FUNCTION_BLOCK VisionCmdProcessor EXTENDS Module
VAR_INPUT
	Command: STRING(GVL.COMMAND_LEN) := '';
	LogicCmdIO: REFERENCE TO ST_LogicCmdIO;
	VisionSystemIpAddress: STRING(19) := '127.0.0.1';
	VisionSystemPort: UINT := 50011;
END_VAR
VAR_OUTPUT
	VisionStateText: STRING := 'READY';
END_VAR
VAR
	_CaptureImage_Output: STRING(255);
	_CaptureImage_WorkerUid: STRING;
	_LocatePart_Output: STRING(255);
	_LocatePart_WorkerUid: STRING;
	_RunCalibration_Output: STRING(255);
	_RunCalibration_WorkerUid: STRING;
	_Vision: OpenCV;
	_VisionCommandParser: ParseVisionCmd;
	_VisionDoneRtrig: R_TRIG;
	_VisionBusyRtrig: R_TRIG;
	_VisionResult: STRING(255);
	_ResultPosition: INT;
	_ResultPosition_CAL: INT;
	_ResultPosition_LOC: INT;
	_ResultPosition_CAP: INT;
	_SpacePosition: INT;
	_VisionObjectIndex: UINT;
	_VisionRatio: REAL;
	_VisionRotation: REAL;
	_VisionError: REAL;
	_PartsCount: UDINT;
	_UnitModeCurrentState: PACK_ML.State;
END_VAR
VAR CONSTANT
	_RESPONSE_CAL: STRING := 'res: CAL ';
	_RESPONSE_LOC: STRING := 'res: LOC ';
	_RESPONSE_CAP: STRING := 'res: CAP ';
	_STEP_DONE: INT := 1000;
	_STEP_IDLE: INT := 0;
	_STEP_COMMAND: INT := 20;
	_STEP_TRIGGER: INT := 30;
	_STEP_WAIT: INT := 40;
	_STEP_ERR: INT := 50;
END_VAR

SUPER^();

// PackML state machine implementation
_UnitModeCurrentState := SUPER^._UnitMode.CurrentState;

//
CASE SUPER^._SeqMain OF
	
    _STEP_DONE:
		SUPER^._SeqMain := _STEP_IDLE;
        
    _STEP_IDLE:
		// hang out here until called to run
        
    _STEP_COMMAND: // parse vision command
        _VisionCommandParser(Command:=Command);
		IF _VisionCommandParser.Error THEN
			SUPER^.M_Error(Description:=_VisionCommandParser.ErrorDescription);
			//
			SUPER^._SeqMain := _STEP_ERR;
		ELSE
			IF _VisionCommandParser.stCommand.Timeout > 0 THEN
				SUPER^._TimeoutTimer.PT := UDINT_TO_TIME(_VisionCommandParser.stCommand.Timeout * 1000);
			END_IF
			//
			SUPER^._SeqMain := _STEP_TRIGGER;
		END_IF
		
	_STEP_TRIGGER: //
		CASE _VisionCommandParser.stCommand.CommandType OF
			DUT_Command_VisionType.Calibrate: //
				_Vision.M_CalibrateCamera(	iImageWidth:= _VisionCommandParser.stCommand.ImageWidth, 
											iImageHeight:= _VisionCommandParser.stCommand.ImageHeight, 
											fCalCheckerSize:= _VisionCommandParser.stCommand.Calibrate.CheckerSize, 
											iCalCheckerX:= _VisionCommandParser.stCommand.Calibrate.CheckerXCount, 
											iCalCheckerY:= _VisionCommandParser.stCommand.Calibrate.CheckerYCount,
                                            uTimeout:=_VisionCommandParser.stCommand.Timeout);
			
			DUT_Command_VisionType.Acquire: //
				_Vision.M_CaptureImage(	iImageWidth:= _VisionCommandParser.stCommand.ImageWidth, 
										iImageHeight:= _VisionCommandParser.stCommand.ImageHeight,
                                        uTimeout:=_VisionCommandParser.stCommand.Timeout);
			
			DUT_Command_VisionType.LocatePart: //
				_PartsCount := 0;
				LogicCmdIO.Register[_VisionCommandParser.stCommand.Locate.ResultPosition] := 0;
				_Vision.M_LocatePart( 	iImageWidth:= _VisionCommandParser.stCommand.ImageWidth, 
										iImageHeight:= _VisionCommandParser.stCommand.ImageHeight, 
										iMaxPos:= _VisionCommandParser.stCommand.Locate.MaxParts, 
										dMaxOverlap:= _VisionCommandParser.stCommand.Locate.MaxOverlap, 
										dScore:= _VisionCommandParser.stCommand.Locate.Score, 
										dToleranceAngle:= _VisionCommandParser.stCommand.Locate.ToleranceAngle,
                                        uTimeout:=_VisionCommandParser.stCommand.Timeout,
										sTemplateName:=_VisionCommandParser.stCommand.Locate.TemplateName,
										sScriptFilename:=_VisionCommandParser.stCommand.Locate.ScriptFilename);
			
		END_CASE;
		
		//
		SUPER^._SeqMain := _STEP_WAIT;
		
	_STEP_WAIT: //
		IF _VisionDoneRtrig.Q THEN
			
			//
			_VisionResult := _Vision.P_Response;
			
			//
			_ResultPosition_CAL := FIND(STR1:=_VisionResult,STR2:=_RESPONSE_CAL);
			_ResultPosition_LOC := FIND(STR1:=_VisionResult,STR2:=_RESPONSE_LOC);
			_ResultPosition_CAP := FIND(STR1:=_VisionResult,STR2:=_RESPONSE_CAP);
			
			//
			IF _ResultPosition_CAL > 0 THEN 
				// calibration was completed
				// res: CAL rat:23.23 rot:23.23 err:23.23
				_VisionResult := MID(STR:=_VisionResult,LEN:=LEN(_VisionResult)-LEN(_RESPONSE_CAL),POS:=LEN(_RESPONSE_CAL)+1);
				//VisionStateText := CONCAT(VisionStateText, '\n');
				//VisionStateText := CONCAT(VisionStateText, _VisionResult);
				// rat:23.23 rot:23.23 err:23.23
				_ResultPosition := FIND(STR1:=_VisionResult,STR2:='rat:');
				IF _ResultPosition > 0 THEN
					_VisionResult := MID(STR:=_VisionResult,LEN:=LEN(_VisionResult)-LEN('rat:'),POS:=LEN('rat:')+1);
					_SpacePosition := FIND(STR1:=_VisionResult,STR2:=' ');
					_VisionRatio := STRING_TO_REAL(MID(STR:=_VisionResult,LEN:=_SpacePosition-1,POS:=1));
					_VisionResult := MID(STR:=_VisionResult,LEN:=LEN(_VisionResult)-_SpacePosition,POS:=_SpacePosition+1);
				END_IF
				// rot:23.23 err:23.23
				_ResultPosition := FIND(STR1:=_VisionResult,STR2:='rot:');
				IF _ResultPosition > 0 THEN
					_VisionResult := MID(STR:=_VisionResult,LEN:=LEN(_VisionResult)-LEN('rot:'),POS:=LEN('rot:')+1);
					_SpacePosition := FIND(STR1:=_VisionResult,STR2:=' ');
					_VisionRotation := STRING_TO_REAL(MID(STR:=_VisionResult,LEN:=_SpacePosition-1,POS:=1));
					_VisionResult := MID(STR:=_VisionResult,LEN:=LEN(_VisionResult)-_SpacePosition,POS:=_SpacePosition+1);
				END_IF
				// err:23.23
				_ResultPosition := FIND(STR1:=_VisionResult,STR2:='err:');
				IF _ResultPosition > 0 THEN
					_VisionResult := MID(STR:=_VisionResult,LEN:=LEN(_VisionResult)-LEN('err:'),POS:=LEN('err:')+1);
					_SpacePosition := FIND(STR1:=_VisionResult,STR2:=' ');
					_VisionError := STRING_TO_REAL(MID(STR:=_VisionResult,LEN:=_SpacePosition-1,POS:=1));
					_VisionResult := MID(STR:=_VisionResult,LEN:=LEN(_VisionResult)-_SpacePosition,POS:=_SpacePosition+1);
				END_IF
				
			ELSIF _ResultPosition_LOC > 0 THEN 
				// part was located
				// 'res: LOC obj:0 cx:54.66 cy:119.45 a:-12.87 s:0.84 $NLOC obj:1 cx:71.49 cy:100.06 a:10.13 s:0.83 $N'
				_VisionResult := MID(STR:=_VisionResult,LEN:=LEN(_VisionResult)-LEN(_RESPONSE_LOC),POS:=LEN(_RESPONSE_LOC)+1);
				//VisionStateText := CONCAT(VisionStateText, '\n');
				//VisionStateText := CONCAT(VisionStateText, _VisionResult);
				_VisionObjectIndex := 0;
				WHILE FIND(STR1:=_VisionResult,STR2:='obj:') > 0 
					AND _VisionObjectIndex <= _VisionCommandParser.stCommand.Locate.MaxParts 
					AND _VisionObjectIndex + _VisionCommandParser.stCommand.Locate.ResultPosition < GVL.VIS_ARR_END DO
					// 'obj:0 cx:54.66 cy:119.45 a:-12.87 s:0.84 $NLOC obj:1 cx:71.49 cy:100.06 a:10.13 s:0.83 $N'
					// $NLOC obj:1 cx:71.49 cy:100.06 a:10.13 s:0.83 $N'
					_ResultPosition := FIND(STR1:=_VisionResult,STR2:='obj:');
					IF _ResultPosition > 0 THEN
						_PartsCount := _PartsCount + 1;
						_VisionResult := MID(STR:=_VisionResult,LEN:=LEN(_VisionResult)-_ResultPosition-LEN('obj:')+1,POS:=_ResultPosition+LEN('obj:'));
						_SpacePosition := FIND(STR1:=_VisionResult,STR2:=' ');
						_VisionObjectIndex := STRING_TO_UINT(MID(STR:=_VisionResult,LEN:=_SpacePosition-1,POS:=1));
						SUPER^.VisionRegisters[_VisionCommandParser.stCommand.Locate.ResultPosition + _VisionObjectIndex].Comment := CONCAT('obj:', UDINT_TO_STRING(_VisionObjectIndex));
						_VisionResult := MID(STR:=_VisionResult,LEN:=LEN(_VisionResult)-_SpacePosition,POS:=_SpacePosition+1);
					END_IF
					// cx:54.66 cy:119.45 a:-12.87 s:0.84 $NLOC obj:1 cx:71.49 cy:100.06 a:10.13 s:0.83 $N'
					_ResultPosition := FIND(STR1:=_VisionResult,STR2:='cx:');
					IF _ResultPosition > 0 THEN
						_VisionResult := MID(STR:=_VisionResult,LEN:=LEN(_VisionResult)-LEN('cx:'),POS:=LEN('cx:')+1);
						_SpacePosition := FIND(STR1:=_VisionResult,STR2:=' ');
						SUPER^.VisionRegisters[_VisionCommandParser.stCommand.Locate.ResultPosition + _VisionObjectIndex].Position.X := STRING_TO_LREAL(MID(STR:=_VisionResult,LEN:=_SpacePosition-1,POS:=1));
						_VisionResult := MID(STR:=_VisionResult,LEN:=LEN(_VisionResult)-_SpacePosition,POS:=_SpacePosition+1);
					END_IF
					// cy:119.45 a:-12.87 s:0.84 $NLOC obj:1 cx:71.49 cy:100.06 a:10.13 s:0.83 $N'
					_ResultPosition := FIND(STR1:=_VisionResult,STR2:='cy:');
					IF _ResultPosition > 0 THEN
						_VisionResult := MID(STR:=_VisionResult,LEN:=LEN(_VisionResult)-LEN('cy:'),POS:=LEN('cy:')+1);
						_SpacePosition := FIND(STR1:=_VisionResult,STR2:=' ');
						SUPER^.VisionRegisters[_VisionCommandParser.stCommand.Locate.ResultPosition + _VisionObjectIndex].Position.Y := STRING_TO_LREAL(MID(STR:=_VisionResult,LEN:=_SpacePosition-1,POS:=1));
						_VisionResult := MID(STR:=_VisionResult,LEN:=LEN(_VisionResult)-_SpacePosition,POS:=_SpacePosition+1);
					END_IF
					// a:-12.87 s:0.84 $NLOC obj:1 cx:71.49 cy:100.06 a:10.13 s:0.83 $N'
					_ResultPosition := FIND(STR1:=_VisionResult,STR2:='a:');
					IF _ResultPosition > 0 THEN
						_VisionResult := MID(STR:=_VisionResult,LEN:=LEN(_VisionResult)-LEN('a:'),POS:=LEN('a:')+1);
						_SpacePosition := FIND(STR1:=_VisionResult,STR2:=' ');
						SUPER^.VisionRegisters[_VisionCommandParser.stCommand.Locate.ResultPosition + _VisionObjectIndex].Position.A := STRING_TO_LREAL(MID(STR:=_VisionResult,LEN:=_SpacePosition-1,POS:=1));
						_VisionResult := MID(STR:=_VisionResult,LEN:=LEN(_VisionResult)-_SpacePosition,POS:=_SpacePosition+1);
					END_IF
					// s:0.84 $NLOC obj:1 cx:71.49 cy:100.06 a:10.13 s:0.83 $N'
					_ResultPosition := FIND(STR1:=_VisionResult,STR2:='s:');
					IF _ResultPosition > 0 THEN
						_VisionResult := MID(STR:=_VisionResult,LEN:=LEN(_VisionResult)-LEN('s:'),POS:=LEN('s:')+1);
						_SpacePosition := FIND(STR1:=_VisionResult,STR2:=' ');
						SUPER^.VisionRegisters[_VisionCommandParser.stCommand.Locate.ResultPosition + _VisionObjectIndex].Scaling := STRING_TO_REAL(MID(STR:=_VisionResult,LEN:=_SpacePosition-1,POS:=1));
						_VisionResult := MID(STR:=_VisionResult,LEN:=LEN(_VisionResult)-_SpacePosition,POS:=_SpacePosition+1);
					END_IF
					// $NLOC obj:1 cx:71.49 cy:100.06 a:10.13 s:0.83 $N'
				END_WHILE
				// return how many part were found
				LogicCmdIO.Register[_VisionCommandParser.stCommand.Locate.ResultPosition] := _PartsCount;
				
			ELSIF _ResultPosition_CAP > 0 THEN 
				// image was captured
				
			END_IF
			
			//
			SUPER^._SeqMain := _STEP_DONE;
			
		END_IF

END_CASE

//
_Vision(sIpAddress:= VisionSystemIpAddress, uPort:= VisionSystemPort);

//
_VisionBusyRtrig(clk:=_Vision.P_Busy);
IF _VisionBusyRtrig.Q THEN
	VisionStateText := 'BUSY';
END_IF

//
_VisionDoneRtrig(clk:=_Vision.P_Done);
IF _VisionDoneRtrig.Q THEN
	VisionStateText := 'DONE.';
	VisionStateText := CONCAT(VisionStateText, ' Found ');
	VisionStateText := CONCAT(VisionStateText, UDINT_TO_STRING(_PartsCount));
	VisionStateText := CONCAT(VisionStateText, ' parts.');
END_IF

METHOD PROTECTED M_Aborting : BOOL
CASE _SeqAborting OF
	0:
		_Vision.M_Cancel();
		_SeqAborting := _SeqAborting + 1;
		
	1: 
		IF NOT _Vision.P_Busy THEN
			SUPER^.M_StateComplete();
			_SeqAborting := 0;
		END_IF
END_CASE
END_METHOD

METHOD PROTECTED M_Complete : BOOL
// once complete, reset to get back to idle
SUPER^._UnitMode.Reset();
END_METHOD

METHOD PROTECTED M_Execute : BOOL
// here we want to execute our commands/jobs/etc and set completed when done.
IF SUPER^._SeqMain =_STEP_IDLE THEN
	SUPER^.M_StateComplete();
END_IF
END_METHOD

METHOD M_ReconnectVisionSystem : BOOL
// TODO may want to make sure the state machine is not in execute?
_Vision.M_Reconnect();
END_METHOD

METHOD PROTECTED M_Resetting : BOOL
CASE SUPER^._SeqResetting OF
	0:
		_Vision.M_Reset();
		_SeqResetting := _SeqResetting + 1;
	1:
		IF NOT _Vision.P_Error THEN
			//VisionStateText := 'RESET';
			SUPER^.M_StateComplete();
			_SeqResetting := 0;
		END_IF
END_CASE
END_METHOD

METHOD PROTECTED M_SetPackML : BOOL
SUPER^._UnitMode(	sName := 'Vision Processor',
				eInitialState := PACK_ML.State.Idle,
				xActive := TRUE);
END_METHOD

METHOD PROTECTED M_Starting : BOOL
// here we want to clear things and get ready for the execute state
// I can consider this the "INIT" state
SUPER^._SeqMain := _STEP_COMMAND;
SUPER^.M_StateComplete();
END_METHOD

{attribute 'monitoring' := 'variable'}
PROPERTY P_PartsCount : REFERENCE TO UDINT
GET
P_PartsCount REF= _PartsCount;
END_GET
END_PROPERTY

{attribute 'monitoring' := 'variable'}
PROPERTY P_VisionSystemConnected : REFERENCE TO BOOL
GET
P_VisionSystemConnected REF= _Vision._TcpClient.bConnected;
END_GET
END_PROPERTY

END_FUNCTION_BLOCK

(* stored: Version 1.1.0.1
   POU VisionCmdProcessor: Id {fe68b725-9761-4240-89f1-03981366ea66}, SpecialFunc None
   Method M_Aborting: Id {d513ea01-4f59-4a93-8842-106eb97fa165}
   Method M_Complete: Id {fcfc6b30-29f1-4c96-9dec-23fe83a707f7}
   Method M_Execute: Id {4fb297bd-99b3-45b8-9db0-a39dde1b30d8}
   Method M_ReconnectVisionSystem: Id {bccf85b8-1449-40b5-9076-7f7a8ac52707}
   Method M_Resetting: Id {62ae2670-1ac3-4949-b0cc-afaf62b4bcb3}
   Method M_SetPackML: Id {93afa927-2608-4b3d-9460-07c2fd48c33a}
   Method M_Starting: Id {02db5f8f-59c2-4bc3-a7b7-0c1db0560d27}
   Property P_PartsCount: Id {59a35101-d609-430e-a7f5-a7dd6d208165}
   Get Get: Id {d3ea4b4b-4335-46ba-9e4d-417107aade88}
   Property P_VisionSystemConnected: Id {095e3029-762d-4123-a2cd-4e83671e3172}
   Get Get: Id {0da79bc0-af22-4674-ae1a-efb3a7b47aa6} *)
